TYPE
    ST_AssemblyStart : STRUCT
        ComponentID : T_MaxString;
    END_STRUCT
END_TYPE

(* stored: Version 1.1.0.1
   DUT ST_AssemblyStart: Id {dd09fe7f-efab-4c51-abb6-a8b7b56730dc} *)
